// TIA Portal V20 export
VAR_GLOBAL   // PLC tag table "LGR_Const_Drive_AxisNo"
END_VAR
VAR_GLOBAL CONSTANT   // user constants
   X : USInt := 1;
   Y : USInt := 2;
   Z : USInt := 3;
   G : USInt := 4;
   X1 : USInt := 5;
   X2 : USInt := 6;
END_VAR
